FUNCTION deg2rad : lreal
VAR_INPUT
	angle_deg:lreal;
END_VAR
VAR
END_VAR

deg2rad:=angle_deg*pi/180;

END_FUNCTION

(* stored: Version 1.1.0.1, ProductVersion 3.1.4024.11
   POU deg2rad: Id {85667c5a-688c-4f76-b165-bfdaa4c9f9b1}, SpecialFunc None *)
